PROGRAM Klant
VAR
	state : KlantToestand;
END_VAR

CASE state OF
	KlantToestand.voorBalie:
		IF GVL.klantWordtGeholpen THEN
			state := klantToestand.wordtGeholpen;
		END_IF
		
	KlantToestand.wordtGeholpen:
		IF GVL.klantWacht THEN
			state := KlantToestand.aanHetWachten;
		END_IF
		
	KlantToestand.aanHetWachten:
		IF GVL.verfAanKlantGegeven THEN
			state := KlantToestand.heeftVerf;
		END_IF
		
	KlantToestand.heeftVerf:
		GVL.klantWiltVerf := FALSE;
END_CASE

END_PROGRAM

(* stored: Version 1.1.0.1, ProductVersion 3.1.4024.15
   POU Klant: Id {83c63601-1ba3-4a51-a444-c63301a380d8}, SpecialFunc None *)
